// TIA Portal V20 export
TYPE "typeEm2MonitoringJobInterface"
// stored: Access Published, Namespace Unit1
   STRUCT
      busyAutoSplice { ExternalWritable := 'False'} : Bool;
      doneAutoSplice { ExternalWritable := 'False'} : Bool;
   END_STRUCT;
END_TYPE
